(* CODESYS project FU_wBitGetPart.xml

Project tree, tasks and I/O mapping:
  function FU_wBitGetPart [ST]
*)

// FU_wBitGetPart
//This function gets only the needed bits of a variable
// |**Version**|**Author**| **Date** |**Changes**
// | 1         | NSN      | 16-03-22 | Creation
FUNCTION FU_wBitGetPart : WORD
VAR_INPUT
	value			:WORD;		//Variable to get value from
	amount			:BYTE;		//Amount of bits to change
	offset			:BYTE;		//Offset in variable to change bits at
END_VAR

FU_wBitGetPart		:=		SHR(value,offset) AND GConstants.binaryMaskWord[amount];

END_FUNCTION
